{attribute 'GeneratedUsingTerminal: EL9540-0010-0016'}
{attribute addProperty BoxType "EL9540-0010-0016"}
{attribute addProperty Id "UndervoltageAT %I*BOOL1OvervoltageAT %I*BOOL1"}
{attribute addProperty CRC "3677696296"}
{attribute addProperty Size "2"}
TYPE Status_Up_DB353128 EXTENDS InputBase_8311D824 :
STRUCT
	{attribute addProperty Name "Undervoltage"}
	Undervoltage AT %I* : BOOL;
	{attribute addProperty Name "Overvoltage"}
	Overvoltage AT %I* : BOOL;
END_STRUCT
END_TYPE

(* stored: Version 1.2.0.0, ProductVersion 3.1.4024.9
   DUT Status_Up_DB353128: Id {a867f03a-81d4-4368-90ed-ddcabb602e39} *)
